(* IEC 61131-3 sources: Industry-PLC-LLM/data/PLCBEAD_repo/PLCBEAD_PLCEmbed-main/PLC-BEAD/Source/GEB/WORD_TO_RANGE, 1 file *)

(* ---- WORD_TO_RANGE.ST ---- *)
FUNCTION _WORD_TO_REAL:REAL
	VAR_INPUT
		IN :	WORD;
	END_VAR
	_WORD_TO_REAL := UINT_TO_REAL(WORD_TO_UINT(IN));
END_FUNCTION

FUNCTION WORD_TO_RANGE:REAL
	VAR_INPUT
		X :	WORD;
		LOW :	REAL;
		HIGH :	REAL;
	END_VAR
	WORD_TO_RANGE := (HIGH - LOW) * _WORD_TO_REAL(X) * 0.00001525902189669640 + low;
END_FUNCTION

PROGRAM program0
  	VAR
		X :	WORD;
		LOW :	REAL;
		HIGH :	REAL;
		CEIL5_OUT : REAL;
	  END_VAR

  	CEIL5_OUT := WORD_TO_RANGE(X, LOW, HIGH);
END_PROGRAM
